RoboDK station: rectangle.rdk

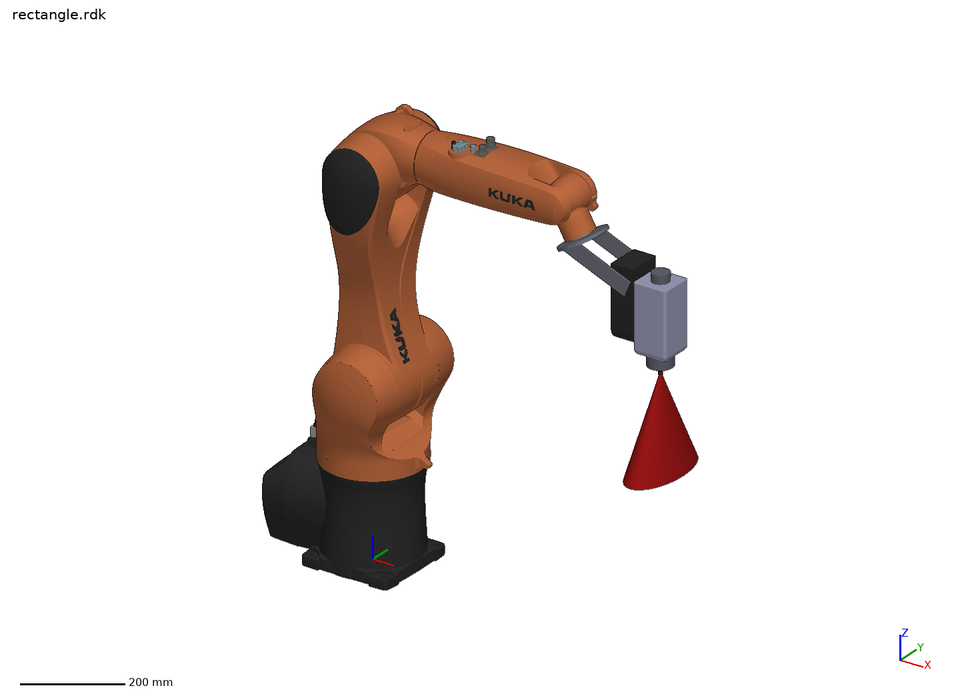
[picture v0: the station drawn from its stored meshes, robots at their saved joint values, targets as dots, program paths as lines]
Station rectangle (saved by RoboDK 5.8.0). Poses are relative to the parent item; angles as X-Y-Z fixed-axis rotations.
  - frame KUKA KR 6 R900 sixx Base at (0, 0, 0) mm
    - robot KUKA KR 6 R900 sixx: 6 axes, payload 6 kg, reach 901 mm, repeatability 0.03 mm, weight 52 kg
        modified DH rows (alpha deg, a mm, theta deg, d mm): 0, 0, 0, 400; -90, 25, 0, 0; 0, 455, -90, 0; -90, 35, 0, 420; 90, 0, 0, 0; -90, 0, 180, 80
        joint limits [-170, -190, -120, -185, -120, -350] to [170, 45, 156, 185, 120, 350]; home [0, -90, 90, 0, 0, 0]; saved at [0, -90, 90, 0, 60, 0]
      - tool Paint gun, TCP at (50, 0, 450) mm, rotated rx 0 ry 30 rz 0 deg, size 203.2 x 279.7 x 471.5 mm
  - Python program rectangle (listed below)
  - program main (1 instructions, listed below)

--- Python program rectangle ---
from robodk.robolink import *  # API to communicate with RoboDK
from robodk.robomath import *  # Basic matrix operations

# Initialize RoboDK API
RDK = Robolink()

# Select a robot (popup displayed if multiple robots are available)
robot = RDK.ItemUserPick('Select a robot', ITEM_TYPE_ROBOT)
if not robot.Valid():
    raise Exception('No robot selected or available')

# Get the current position of the TCP with respect to the reference frame
target_ref = robot.Pose()
pos_ref = target_ref.Pos()
print("Drawing a rectangle around the target: ")
print(Pose_2_TxyzRxyz(target_ref))

# Move the robot to the starting point
robot.MoveJ(target_ref)

# Set reference and tool frames
robot.setPoseFrame(robot.PoseFrame())
robot.setPoseTool(robot.PoseTool())
robot.setRounding(10)  # Set blending radius
robot.setSpeed(200)  # Set linear speed in mm/s

# rectangle parameters
side_length = 200  # Length of each side of the rectangle
rectangle_points = [
    (side_length / 2, side_length ),  # Top-right corner
    (-side_length / 2, side_length ),  # Top-left corner
    (-side_length / 2, -side_length ),  # Bottom-left corner
    (side_length / 2, -side_length )   # Bottom-right corner
]

# Loop through the rectangle vertices
for i, (dx, dy) in enumerate(rectangle_points + [rectangle_points[0]]):  # Close the rectangle
    # Calculate the new position
    target_i = Mat(target_ref)  # Copy the reference pose
    pos_i = target_i.Pos()  # Extract position from the reference pose
    pos_i[0] += dx  # Update X coordinate
    pos_i[1] += dy  # Update Y coordinate
    target_i.setPos(pos_i)  # Set the updated position

    # Move the robot to the calculated vertex
    print(f"Moving to vertex {i + 1}: dx={dx}, dy={dy}")
    print(Pose_2_TxyzRxyz(target_i))
    robot.MoveL(target_i)

# Return to the center position
robot.MoveL(target_ref)

print("rectangle drawing complete!")

--- program main (robot KUKA KR 6 R900 sixx) ---
  Call rectangle
